// TIA Portal project "ejercicio2" (V15.1)

(* hardware
DEVICE "HMI_1"  KTP700 Basic PN
   slot 0: "HMI_1"  KTP700 Basic PN  6AV2 123-2GB03-0AX0  15.1.0.0
   slot 1: "HMI_RT_1"  KTP700 Basic PN  6AV2 123-2GB03-0AX0  15.1.0.0
   slot 5: "HMI_1.IE_CP_1"  PROFINET Interface  15.0.1.0
      slot 1: "Interfaz PROFINET_1"  PROFINET Interface
         slot 1: "Port_1"  Port
DEVICE "S7-1200 station_1"  S7-1200 Station
   slot 0: "Rack_0"  S7-1200 Rack  Rack  V1.0
   slot 1: "PLC_1"  CPU 1215C AC/DC/Rly  6ES7 215-1BG40-0XB0  V4.2
*)

// ===== PLC "PLC_1"  CPU 1215C AC/DC/Rly =====

VAR_GLOBAL   // PLC tag table "Tabla de variables estándar"
   "q1" AT %M0.0 : Bool;   // estado 1
   "q2" AT %M0.1 : Bool;   // estado 2
   "q3b" AT %M0.2 : Bool;   // estado 3b
   "q3c" AT %M0.3 : Bool;   // estado 3c
   "q4b" AT %M0.4 : Bool;   // estado 4b
   "q4c" AT %M0.5 : Bool;   // estado 4c
   "A" AT %M1.0 : Bool;   // cinta A
   "B" AT %M1.1 : Bool;   // cinta B
   "C" AT %M1.2 : Bool;   // cinta C
   "P1" AT %M1.3 : Bool;   // piston 1
   "P2" AT %M1.4 : Bool;   // piston 2
   "P3" AT %M1.5 : Bool;   // piston 3
   "CP" AT %M2.0 : Bool;   // caja grande
   "CG" AT %M2.1 : Bool;   // caja pequeña
   "S1" AT %M2.2 : Bool;   // sensor 1
   "S2" AT %M2.3 : Bool;   // sensor 2
   "S3" AT %M2.4 : Bool;   // sensor3
END_VAR

ORGANIZATION_BLOCK "Main"   // OB1, LAD, ProgramCycle
TITLE = "Main Program Sweep (Cycle)"
{ S7_Optimized_Access := 'TRUE' }
VERSION : 0.1
   VAR_INPUT
      Initial_Call : Bool;   // Initial call of this OB
      Remanence : Bool;   // =True, if remanent data are available
   END_VAR
   VAR_TEMP   // added for the SCL form of the ladder/FBD networks
      _w1 : Bool;
   END_VAR
BEGIN

REGION Network 1: seteamos estado 1 como inicial
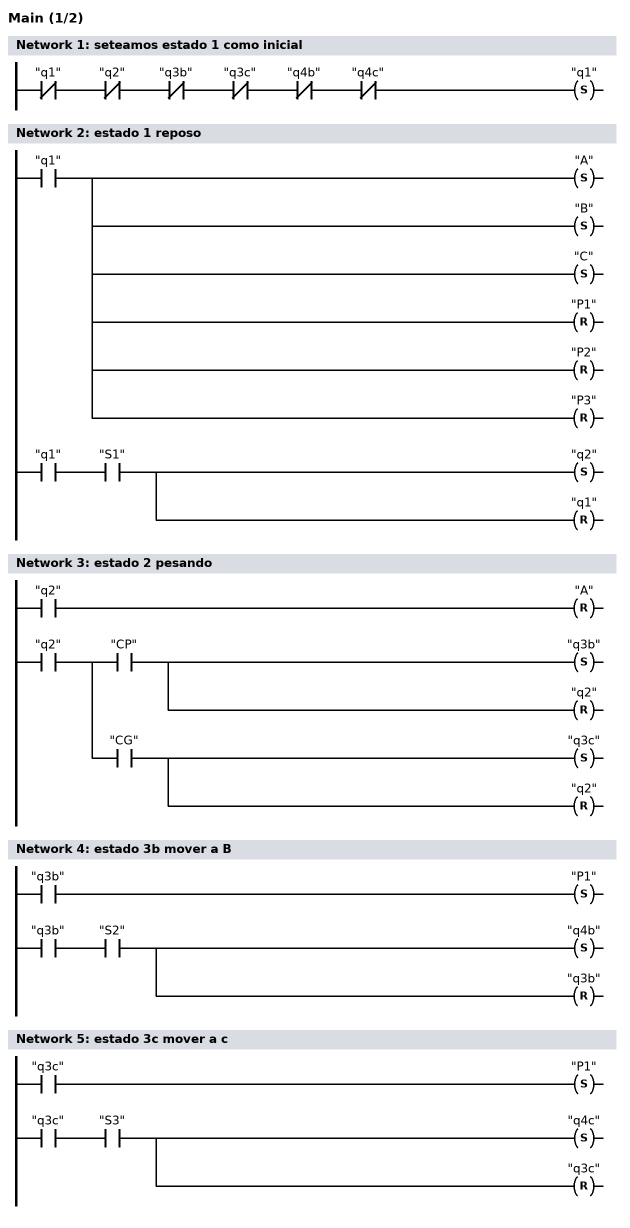
   RUNG wire#powerrail
      I_Contact( "q1" )
      I_Contact( "q2" )
      I_Contact( "q3b" )
      I_Contact( "q3c" )
      I_Contact( "q4b" )
      I_Contact( "q4c" )
      S_Coil( "q1" )
   END_RUNG
   // the same network as SCL:
   IF NOT "q1" AND NOT "q2" AND NOT "q3b" AND NOT "q3c" AND NOT "q4b" AND NOT "q4c" THEN
       "q1" := TRUE;
   END_IF;
END_REGION

REGION Network 2: estado 1 reposo
   RUNG wire#powerrail
      Contact( "q1" )
      wire#w1
      S_Coil( "A" )
   END_RUNG
   RUNG wire#w1
      S_Coil( "B" )
   END_RUNG
   RUNG wire#w1
      S_Coil( "C" )
   END_RUNG
   RUNG wire#w1
      R_Coil( "P1" )
   END_RUNG
   RUNG wire#w1
      R_Coil( "P2" )
   END_RUNG
   RUNG wire#w1
      R_Coil( "P3" )
   END_RUNG
   RUNG wire#powerrail
      Contact( "q1" )
      Contact( "S1" )
      wire#w2
      S_Coil( "q2" )
   END_RUNG
   RUNG wire#w2
      R_Coil( "q1" )
   END_RUNG
   // the same network as SCL:
   IF "q1" THEN
       "A" := TRUE;
       "B" := TRUE;
       "C" := TRUE;
       "P1" := FALSE;
       "P2" := FALSE;
       "P3" := FALSE;
   END_IF;
   IF "q1" AND "S1" THEN
       "q2" := TRUE;
       "q1" := FALSE;
   END_IF;
END_REGION

REGION Network 3: estado 2 pesando
   RUNG wire#powerrail
      Contact( "q2" )
      R_Coil( "A" )
   END_RUNG
   RUNG wire#powerrail
      Contact( "q2" )
      wire#w1
      Contact( "CP" )
      wire#w2
      S_Coil( "q3b" )
   END_RUNG
   RUNG wire#w2
      R_Coil( "q2" )
   END_RUNG
   RUNG wire#w1
      Contact( "CG" )
      wire#w3
      S_Coil( "q3c" )
   END_RUNG
   RUNG wire#w3
      R_Coil( "q2" )
   END_RUNG
   // the same network as SCL:
   IF "q2" THEN "A" := FALSE; END_IF;
   IF "q2" AND "CP" THEN "q3b" := TRUE; END_IF;
   #_w1 := "q2";
   IF "q2" AND "CP" THEN "q2" := FALSE; END_IF;
   IF #_w1 AND "CG" THEN
       "q3c" := TRUE;
       "q2" := FALSE;
   END_IF;
END_REGION

REGION Network 4: estado 3b mover a B
   RUNG wire#powerrail
      Contact( "q3b" )
      S_Coil( "P1" )
   END_RUNG
   RUNG wire#powerrail
      Contact( "q3b" )
      Contact( "S2" )
      wire#w1
      S_Coil( "q4b" )
   END_RUNG
   RUNG wire#w1
      R_Coil( "q3b" )
   END_RUNG
   // the same network as SCL:
   IF "q3b" THEN "P1" := TRUE; END_IF;
   IF "q3b" AND "S2" THEN
       "q4b" := TRUE;
       "q3b" := FALSE;
   END_IF;
END_REGION

REGION Network 5: estado 3c mover a c
   RUNG wire#powerrail
      Contact( "q3c" )
      S_Coil( "P1" )
   END_RUNG
   RUNG wire#powerrail
      Contact( "q3c" )
      Contact( "S3" )
      wire#w1
      S_Coil( "q4c" )
   END_RUNG
   RUNG wire#w1
      R_Coil( "q3c" )
   END_RUNG
   // the same network as SCL:
   IF "q3c" THEN "P1" := TRUE; END_IF;
   IF "q3c" AND "S3" THEN
       "q4c" := TRUE;
       "q3c" := FALSE;
   END_IF;
END_REGION

REGION Network 6: estado 4b encintar en b
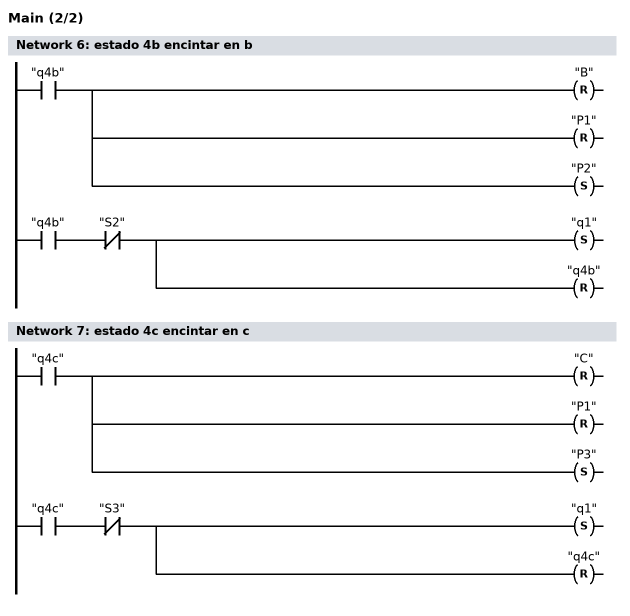
   RUNG wire#powerrail
      Contact( "q4b" )
      wire#w1
      R_Coil( "B" )
   END_RUNG
   RUNG wire#w1
      R_Coil( "P1" )
   END_RUNG
   RUNG wire#w1
      S_Coil( "P2" )
   END_RUNG
   RUNG wire#powerrail
      Contact( "q4b" )
      I_Contact( "S2" )
      wire#w2
      S_Coil( "q1" )
   END_RUNG
   RUNG wire#w2
      R_Coil( "q4b" )
   END_RUNG
   // the same network as SCL:
   IF "q4b" THEN
       "B" := FALSE;
       "P1" := FALSE;
       "P2" := TRUE;
   END_IF;
   IF "q4b" AND NOT "S2" THEN
       "q1" := TRUE;
       "q4b" := FALSE;
   END_IF;
END_REGION

REGION Network 7: estado 4c encintar en c
   RUNG wire#powerrail
      Contact( "q4c" )
      wire#w1
      R_Coil( "C" )
   END_RUNG
   RUNG wire#w1
      R_Coil( "P1" )
   END_RUNG
   RUNG wire#w1
      S_Coil( "P3" )
   END_RUNG
   RUNG wire#powerrail
      Contact( "q4c" )
      I_Contact( "S3" )
      wire#w2
      S_Coil( "q1" )
   END_RUNG
   RUNG wire#w2
      R_Coil( "q4c" )
   END_RUNG
   // the same network as SCL:
   IF "q4c" THEN
       "C" := FALSE;
       "P1" := FALSE;
       "P3" := TRUE;
   END_IF;
   IF "q4c" AND NOT "S3" THEN
       "q1" := TRUE;
       "q4c" := FALSE;
   END_IF;
END_REGION
END_ORGANIZATION_BLOCK

(* ===== HMI "HMI_RT_1" =====
system functions are stored by id; their names below are inferred from use
connection "HMI_Conexión_1": ETHERNET, SMART_S7_1200_OMS

HMI tags "Tabla de variables estándar"
   "Número_imagen_variable" : UInt, internal
   "A" : Bool = PLC A AT %M1.0, 1 s
   "B" : Bool = PLC B AT %M1.1, 1 s
   "C" : Bool = PLC C AT %M1.2, 1 s
   "P1" : Bool = PLC P1 AT %M1.3, 1 s
   "P2" : Bool = PLC P2 AT %M1.4, 1 s
   "P3" : Bool = PLC P3 AT %M1.5, 1 s
   "q1" : Bool = PLC q1 AT %M0.0, 1 s
   "q2" : Bool = PLC q2 AT %M0.1, 1 s
   "q3b" : Bool = PLC q3b AT %M0.2, 1 s
   "q3c" : Bool = PLC q3c AT %M0.3, 1 s
   "q4b" : Bool = PLC q4b AT %M0.4, 1 s
   "q4c" : Bool = PLC q4c AT %M0.5, 1 s
   "S1" : Bool = PLC S1 AT %M2.2, 1 s
   "S2" : Bool = PLC S2 AT %M2.3, 1 s
   "S3" : Bool = PLC S3 AT %M2.4, 1 s
   "CP" : Bool = PLC CP AT %M2.0, 1 s
   "CG" : Bool = PLC CG AT %M2.1, 1 s

text list "Nombre_imagen_lista_texto": 1 'Imagen raíz'

Template "Plantilla_1" 800x480
   Button "Salir" at 714,429 size 71x50; TextOff 'Salir'; PictureOff "ExitRuntime_KTP700_Basic_PN_TR"; PictureOn "ExitRuntime_KTP700_Basic_PN_TR"
      on Release: StopRuntime(0)
   Button "Template_Button" at 614,429 size 71x50; TextOff 'Text'
   Button "Template_Button_1" at 514,429 size 71x50; TextOff 'Text'
   Button "Template_Button_2" at 414,429 size 71x50; TextOff 'Text'
   Button "Template_Button_3" at 314,429 size 71x50; TextOff 'Text'
   Button "Template_Button_4" at 214,429 size 71x50; TextOff 'Text'
   Button "Avisos" at 114,429 size 71x50; TextOff 'Avisos'; PictureOff "AlarmDisplay_KTP700_Basic_PN_TR"; PictureOn "AlarmDisplay_KTP700_Basic_PN_TR"
      on Release: function_ef3f5d25("Ventana de avisos_no_acusado", -1)
   Button "Imagen inicial" at 14,429 size 71x50; TextOff 'Imagen inicial'; PictureOff "NavigateHome_KTP700_Basic_PN_TR"; PictureOn "NavigateHome_KTP700_Basic_PN_TR"
      on Release: ActivateScreen("Imagen raíz", 0)
   SymbolicIOField "Imagen_campo_ES_simbólico" at 93,9 size 600x33; TextOff '0'; TextOn '1'; TextList "Nombre_imagen_lista_texto"
      ProcessValue <- "Número_imagen_variable"
      on Change: ActivateScreenByNumber("Número_imagen_variable", 0)
   DateTimeField "HmiScreenItemData" at 695,25 size 105x25
   DateTimeField "HmiScreenItemData_1" at 695,0 size 105x25
   GraphicView "Logotipo" at 0,0 size 91x51; Picture "Logotipo de HMI_1"

screen "Imagen raíz" 800x480, template "Plantilla_1"
   on GenerateScreen: SetTag("Número_imagen_variable", 1)
   GraphicIOField "PlotLight_Square_G" at 733,55 size 50x50; PictureOn "PilotLight_Square_G_On_256c"; PictureOff "PilotLight_Square_G_Off_256c"
      ProcessValue <- "q1"
   GraphicIOField "PlotLight_Square_G_1" at 733,112 size 50x50; PictureOff "PilotLight_Square_G_Off_256c"; PictureOn "PilotLight_Square_G_On_256c"
      ProcessValue <- "q2"
   GraphicIOField "PlotLight_Square_G_2" at 733,176 size 50x50; PictureOff "PilotLight_Square_G_Off_256c"; PictureOn "PilotLight_Square_G_On_256c"
      ProcessValue <- "q3b"
   GraphicIOField "PlotLight_Square_G_3" at 733,237 size 50x50; PictureOn "PilotLight_Square_G_On_256c"; PictureOff "PilotLight_Square_G_Off_256c"
      ProcessValue <- "q3c"
   GraphicIOField "PlotLight_Square_G_4" at 733,296 size 50x50; PictureOff "PilotLight_Square_G_Off_256c"; PictureOn "PilotLight_Square_G_On_256c"
      ProcessValue <- "q4b"
   GraphicIOField "PlotLight_Square_G_5" at 733,356 size 50x50; PictureOff "PilotLight_Square_G_Off_256c"; PictureOn "PilotLight_Square_G_On_256c"
      ProcessValue <- "q4c"
   GraphicIOField "PlotLight_Round_R_5" at 201,133 size 50x50; PictureOff "PilotLight_Round_R_Off_256c"; PictureOn "PilotLight_Round_R_On_256c"
      ProcessValue <- "C"
   GraphicIOField "PlotLight_Round_R_1" at 113,133 size 50x50; PictureOn "PilotLight_Round_R_On_256c"; PictureOff "PilotLight_Round_R_Off_256c"
      ProcessValue <- "B"
   GraphicIOField "PlotLight_Round_R_2" at 25,133 size 50x50; PictureOn "PilotLight_Round_R_On_256c"; PictureOff "PilotLight_Round_R_Off_256c"
      ProcessValue <- "A"
   GraphicIOField "PlotLight_Round_N_Mono" at 299,133 size 50x50; PictureOn "PilotLight_Round_N_On_mono"; PictureOff "PilotLight_Round_N_Off_mono"
      ProcessValue <- "P1"
   GraphicIOField "PlotLight_Round_N_Mono_1" at 475,133 size 50x50; PictureOff "PilotLight_Round_N_Off_mono"; PictureOn "PilotLight_Round_N_On_mono"
      ProcessValue <- "P3"
   GraphicIOField "PlotLight_Round_N_Mono_2" at 387,133 size 50x50; PictureOff "PilotLight_Round_N_Off_mono"; PictureOn "PilotLight_Round_N_On_mono"
      ProcessValue <- "P2"
   Button "Botón_1" at 25,285 size 70x57; TextOff 'S1'
      Appearance <- "S1"
      on Press: SetBit("S1")
      on Release: ResetBit("S1")
   TextField "Campo de texto_1" at 656,67 size 65x23; Text 'Reposo'
   TextField "Campo de texto_2" at 647,121 size 74x23; Text 'Pesando'
   TextField "Campo de texto_3" at 572,185 size 149x23; Text 'Moviendo hasta B'
   TextField "Campo de texto_4" at 572,250 size 149x23; Text 'Moviendo hasta C'
   TextField "Campo de texto_5" at 585,304 size 136x23; Text 'Encintando en B'
   TextField "Campo de texto_6" at 585,365 size 136x23; Text 'Encintando en C'
   Button "Botón_2" at 140,285 size 70x57; TextOff 'S2'
      on Click: InvertBit("S2")
      Appearance <- "S2"
   Button "Botón_3" at 255,285 size 70x57; TextOff 'S3'
      on Click: InvertBit("S3")
      Appearance <- "S3"
   Button "Botón_4" at 370,285 size 70x57; TextOff 'CP'
      Appearance <- "CP"
      on Press: SetBit("CP")
      on Release: ResetBit("CP")
   Button "Botón_5" at 485,285 size 70x57; TextOff 'CG'
      Appearance <- "CG"
      on Press: SetBit("CG")
      on Release: ResetBit("CG")
   TextField "Campo de texto_7" at 39,188 size 17x23; Text 'A'
   TextField "Campo de texto_8" at 127,188 size 16x23; Text 'B'
   TextField "Campo de texto_9" at 215,188 size 16x23; Text 'C'
   TextField "Campo de texto_10" at 311,187 size 26x23; Text 'P1'
   TextField "Campo de texto_11" at 397,185 size 26x23; Text 'P2'
   TextField "Campo de texto_12" at 490,188 size 26x23; Text 'P3'
   TextField "Campo de texto_13" at 105,98 size 56x23; Text 'Cintas'
   TextField "Campo de texto_14" at 381,98 size 74x23; Text 'Pistones'
*)